TEXTLIST TL_ConnectionDiag
  0 = 'Without Errors'
  1 = 'Invalid Command'
  2 = 'Unknown Command'
  3 = 'Invalid Connection ID'
  4 = 'Invalid CRC'
  5 = 'Watchdog Time Elapsed'
  6 = 'Invalid FSo EAddress'
  7 = 'Invalid Data'
  8 = 'Invalid Comm Param Length'
  9 = 'Invalid Comm Params'
  10 = 'Invalid User Param Length'
  11 = 'Invalid User Params'
  12 = 'FSoE Master Reset\t'
  13 = 'Module Error'
  14 = 'EL290x Error'
  15 = 'Slave Not Yet Started'
   = ''
END_TEXTLIST

(* stored: Version 1.1.0.1, ProductVersion 3.1.4022.12
   TextList TL_ConnectionDiag: Id {9c6bab81-b383-48e8-adeb-cbce92fce396} *)
